// TIA Portal project "AvvioTemporizzatoEV" (V20)

(* hardware
DEVICE "S7-1200 station_1"  S7-1200 Station
   slot 0: "Rack_0"  S7-1200 Rack  Rack  V1.0
   slot 1: "Playground_PLC"  CPU 1214C DC/DC/DC  6ES7 214-1AG40-0XB0  V4.7
   slot 3: "AQ 1x12BIT_1"  AQ1 signal board  6ES7 232-4HA30-0XB0  V1.0
*)

// ===== PLC "Playground_PLC"  CPU 1214C DC/DC/DC =====

VAR_GLOBAL   // PLC tag table "Default tag table"
   "P1" AT %M0.0 : Bool;
   "P2" AT %M0.1 : Bool;
   "START" AT %M0.2 : Bool;
   "START_V1" AT %M0.3 : Bool;
   "START_V2" AT %M0.4 : Bool;
   "START_V3" AT %M0.5 : Bool;
   "STOP_V1" AT %M0.6 : Bool;
   "STOP_V2" AT %M0.7 : Bool;
   "STOP_V3" AT %M1.0 : Bool;
   "EV1_OUT" AT %M1.1 : Bool;
   "EV2_OUT" AT %M1.2 : Bool;
   "EV3_OUT" AT %M1.3 : Bool;
END_VAR

DATA_BLOCK "EV_TIMERS"   // DB1
{ S7_Optimized_Access := 'TRUE' }
VERSION : 0.1
   VAR
      TIMER_V1 : Time := T#5S;
      TIMER_V2 : Time := T#7S;
      TIMER_V3 : Time := T#9S;
   END_VAR
BEGIN
END_DATA_BLOCK

DATA_BLOCK "EV_CONTROL_DB_1"   // DB5
{ S7_Optimized_Access := 'TRUE' }
VERSION : 0.1
// stored: InstanceOfName EV_CONTROL
"EV_CONTROL"
BEGIN
END_DATA_BLOCK

DATA_BLOCK "EV_CONTROL_DB_2"   // DB9
{ S7_Optimized_Access := 'TRUE' }
VERSION : 0.1
// stored: InstanceOfName EV_CONTROL
"EV_CONTROL"
BEGIN
END_DATA_BLOCK

DATA_BLOCK "EV_CONTROL_DB_3"   // DB10
{ S7_Optimized_Access := 'TRUE' }
VERSION : 0.1
// stored: InstanceOfName EV_CONTROL
"EV_CONTROL"
BEGIN
END_DATA_BLOCK

FUNCTION_BLOCK "EV_CONTROL"   // FB1, LAD
{ S7_Optimized_Access := 'TRUE' }
VERSION : 0.1
   VAR_INPUT
      START : Bool;
      STOP : Bool;
      "TIMER" : Time;
   END_VAR
   VAR_OUTPUT
      EV_OUT : Bool;
   END_VAR
   VAR
      ELAPSED : Bool;
      IEC_Timer_0_Instance : TON_TIME;
   END_VAR
   VAR_TEMP
      HELPER_1 : Bool;
   END_VAR
   VAR_TEMP   // added for the SCL form of the ladder/FBD networks
      _w1 : Bool;
      _w2 : Bool;
   END_VAR
BEGIN

REGION Network 1
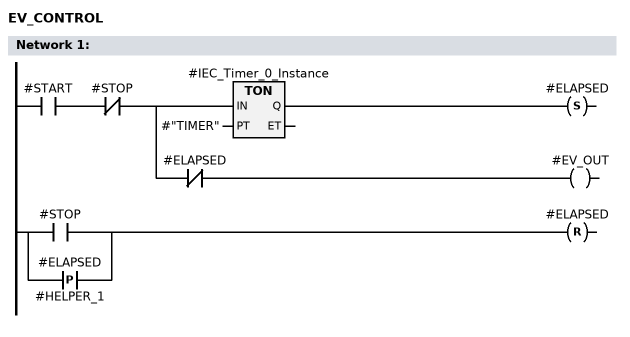
   #_w1 := #START AND NOT #STOP;
   #IEC_Timer_0_Instance(IN := #_w1, PT := #"TIMER");   // TON
   IF #IEC_Timer_0_Instance.Q THEN #ELAPSED := TRUE; END_IF;
   #EV_OUT := #_w1 AND NOT #ELAPSED;
   #_w2 := #ELAPSED AND NOT #HELPER_1;   // rising edge of #ELAPSED
   #HELPER_1 := #ELAPSED;
   IF #STOP OR #_w2 THEN #ELAPSED := FALSE; END_IF;
END_REGION
END_FUNCTION_BLOCK

FUNCTION "AVVIO" : Void   // FC1, LAD
{ S7_Optimized_Access := 'TRUE' }
VERSION : 0.1
   VAR_INPUT
      P1 : Bool;
      P2 : Bool;
   END_VAR
   VAR_OUTPUT
      START : Bool;
   END_VAR
BEGIN

REGION Network 1
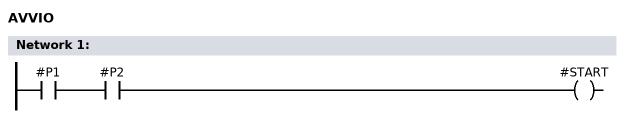
   RUNG wire#powerrail
      Contact( #P1 )
      Contact( #P2 )
      Coil( #START )
   END_RUNG
   // the same network as SCL:
   #START := #P1 AND #P2;
END_REGION
END_FUNCTION

ORGANIZATION_BLOCK "Main"   // OB1, LAD, ProgramCycle
TITLE = "Main Program Sweep (Cycle)"
{ S7_Optimized_Access := 'TRUE' }
VERSION : 0.1
   VAR_INPUT
      Initial_Call : Bool;   // Initial call of this OB
      Remanence : Bool;   // =True, if remanent data are available
   END_VAR
   VAR_TEMP   // added for the SCL form of the ladder/FBD networks
      _w1 : Bool;
   END_VAR
BEGIN

REGION Network 1
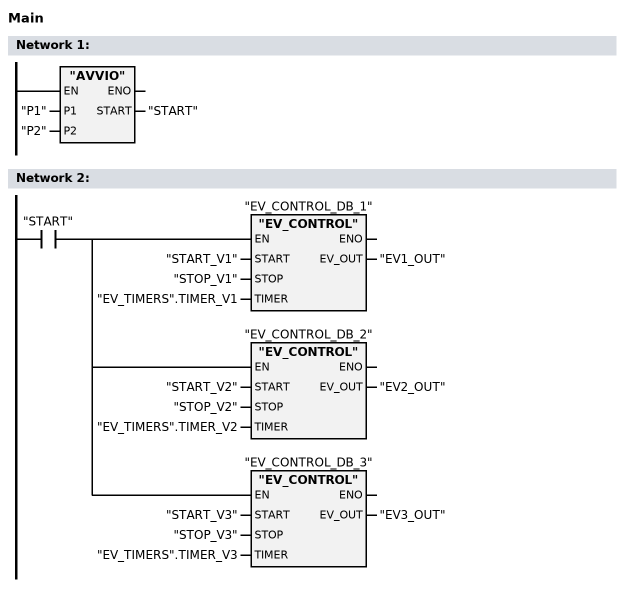
   RUNG wire#powerrail
      "AVVIO"(P1 := "P1", P2 := "P2", START => "START")
   END_RUNG
   // the same network as SCL:
   "AVVIO"(P1 := "P1", P2 := "P2", START => "START");
END_REGION

REGION Network 2
   RUNG wire#powerrail
      Contact( "START" )
      wire#w1
      "EV_CONTROL_DB_1"(START := "START_V1", STOP := "STOP_V1", "TIMER" := "EV_TIMERS".TIMER_V1, EV_OUT => "EV1_OUT")
   END_RUNG
   RUNG wire#w1
      "EV_CONTROL_DB_2"(START := "START_V2", STOP := "STOP_V2", "TIMER" := "EV_TIMERS".TIMER_V2, EV_OUT => "EV2_OUT")
   END_RUNG
   RUNG wire#w1
      "EV_CONTROL_DB_3"(START := "START_V3", STOP := "STOP_V3", "TIMER" := "EV_TIMERS".TIMER_V3, EV_OUT => "EV3_OUT")
   END_RUNG
   // the same network as SCL:
   #_w1 := "START";
   IF #_w1 THEN
       "EV_CONTROL_DB_1"(START := "START_V1",   // "EV_CONTROL"
                         STOP := "STOP_V1",
                         "TIMER" := "EV_TIMERS".TIMER_V1,
                         EV_OUT => "EV1_OUT");
       "EV_CONTROL_DB_2"(START := "START_V2",   // "EV_CONTROL"
                         STOP := "STOP_V2",
                         "TIMER" := "EV_TIMERS".TIMER_V2,
                         EV_OUT => "EV2_OUT");
       "EV_CONTROL_DB_3"(START := "START_V3",   // "EV_CONTROL"
                         STOP := "STOP_V3",
                         "TIMER" := "EV_TIMERS".TIMER_V3,
                         EV_OUT => "EV3_OUT");
   END_IF;
END_REGION
END_ORGANIZATION_BLOCK